FUNCTION_BLOCK T_RoboConnect_SetDigitalOutputTimeout_Fails EXTENDS T_UnitTestBase
VAR
  robot : I_RoboConnect;
  timeOutTimer : TON;
  targetDO : UINT;
  myTestState, prevState :
    (INIT, ARRANGE, ACT, ASSERT) := INIT;
  expected, actual : BOOL;
  counter : UINT;
  returnedTask : I_Task;
END_VAR

CASE myTestState OF
  INIT:
    StateChanged();
    myTestState := ARRANGE;

  ARRANGE:
    IF StateChanged() THEN
      expected := TRUE;
      robot.Connect();
    END_IF

    IF robot.Connected THEN
      myTestState := ACT;
    END_IF

  ACT:
    robot.SetDigitalOutput(targetDO,TRUE, task => returnedTask);
    myTestState := ASSERT;

  ASSERT:
    IF timeOutTimer.Q THEN
      actual := returnedTask.Timeout;
      assertion.AssertEquals_BOOL(expected, actual, 'actual := returnedTask.Timeout');
      TestFinished();
      myTestState := INIT;

    END_IF

END_CASE

robot.CyclicLogic();
timeOutTimer(IN := myTestState = ASSERT);

METHOD FB_init : BOOL
VAR_INPUT
  bInitRetains : BOOL; // if TRUE, the retain variables are initialized (warm start / cold start)
  bInCopyCode : BOOL; // if TRUE, the instance afterwards gets moved into the copy code (online change)
  TestSuite : tcl_SimpleUnitTestLibrary.I_TestSuite;
  robot : I_TcRobot;
  targetDo : UINT;
  timeout : TIME;
END_VAR
THIS^.robot := robot;
THIS^.timeoutTimer.PT := timeout;
THIS^.targetDo := targetDo;
END_METHOD

METHOD PRIVATE StateChanged : BOOL
IF  myTestState = prevState THEN
  RETURN;
END_IF

prevState := myTestState;
StateChanged := TRUE;
END_METHOD

METHOD WaitForCycles : BOOL
VAR_INPUT
  maxCount : UINT;
END_VAR
counter := counter + 1;

IF counter = maxCount THEN
  counter := 0;
  WaitForCycles := TRUE;
END_IF
END_METHOD

END_FUNCTION_BLOCK

(* stored: Version 1.1.0.1
   POU T_TcRobot_SetDigitalOutputTimeout_Fails: Id {eafb8375-49a7-415d-8bdd-afb5ab38b266}, SpecialFunc None
   Method FB_init: Id {eeeb9097-f1e3-440c-a007-90f115ffd194}
   Method StateChanged: Id {66f342fa-56e8-42b2-ac55-f13e4d8cf29b}
   Method WaitForCycles: Id {b8252a2c-559e-42ff-878b-c3696134d473} *)
